(* IEC 61131-3 sources: CodesysTest/export/Interfaces/IComponent.itf, 3 files *)

(* ---- MakeReady.m.st ---- *)
(*#-#-#-#-#-#-#-#-#-#---Declaration---#-#-#-#-#-#-#-#-#-#-#-#-#*)

METHOD MakeReady : BOOL
VAR_INPUT
END_VAR

(* ---- Reset.m.st ---- *)
(*#-#-#-#-#-#-#-#-#-#---Declaration---#-#-#-#-#-#-#-#-#-#-#-#-#*)

METHOD Reset
VAR_INPUT
END_VAR

(* ---- SterilizeVariables.m.st ---- *)
(*#-#-#-#-#-#-#-#-#-#---Declaration---#-#-#-#-#-#-#-#-#-#-#-#-#*)

METHOD SterilizeVariables : BOOL
VAR_INPUT
END_VAR
